// Mitsubishi GX Works2 project: StartStopStepper   PLC: FX2N/FX2NC

PROGRAM MAIN
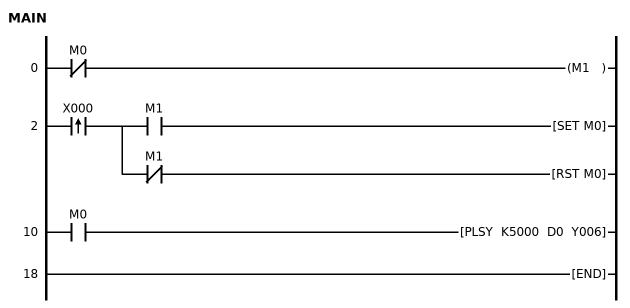
0     LDI     M0
      OUT     M1
2     LDP     X000
      MPS
      AND     M1
      SET     M0
      MPP
      ANI     M1
      RST     M0
10    LD      M0
      PLSY    K5000 D0 Y006
18    END
END_PROGRAM
